// TIA Portal project "thuc_hanh_2" (V14)

(* hardware
DEVICE "S7-1200 station_1"  S7-1200 Station
   slot 0: "Rack_0"  S7-1200 Rack  Rack  V1.0
   slot 1: "PLC_1"  CPU 1214C DC/DC/DC  6ES7 214-1AG40-0XB0  V4.2
*)

// ===== PLC "PLC_1"  CPU 1214C DC/DC/DC =====

VAR_GLOBAL   // PLC tag table "Default tag table"
   "Tag_1" AT %M0.0 : Bool;
   "Tag_2" AT %Q0.0 : Bool;
   "enable" AT %M0.1 : Bool;
   "count_" AT %M0.2 : Bool;
   "reset_count" AT %M0.3 : Bool;
   "done_count" AT %M0.4 : Bool;
   "stop" AT %M0.5 : Bool;
   "Tag_3" AT %Q0.1 : Bool;
   "reset" AT %I0.0 : Bool;
   "start" AT %I0.1 : Bool;
   "Tag_4" AT %I0.3 : Bool;
END_VAR

// folder: System blocks/Program resources

DATA_BLOCK "IEC_Timer_0_DB"   // DB1
{ S7_Optimized_Access := 'TRUE' }
AUTHOR : Simatic
FAMILY : IEC
NAME : IEC_TMR
VERSION : 1.0
// stored: InstanceOfName IEC_TIMER
"IEC_TIMER"
BEGIN
END_DATA_BLOCK

DATA_BLOCK "IEC_Timer_0_DB_1"   // DB2
{ S7_Optimized_Access := 'TRUE' }
AUTHOR : Simatic
FAMILY : IEC
NAME : IEC_TMR
VERSION : 1.0
// stored: InstanceOfName IEC_TIMER
"IEC_TIMER"
BEGIN
END_DATA_BLOCK

DATA_BLOCK "IEC_Counter_0_DB"   // DB3
{ S7_Optimized_Access := 'TRUE' }
AUTHOR : Simatic
FAMILY : IEC
NAME : CNTR
VERSION : 1.0
// stored: InstanceOfName IEC_COUNTER
"IEC_COUNTER"
BEGIN
END_DATA_BLOCK

// folder: (top level)

ORGANIZATION_BLOCK "Main"   // OB1, LAD, ProgramCycle
TITLE = "Main Program Sweep (Cycle)"
{ S7_Optimized_Access := 'TRUE' }
VERSION : 0.1
   VAR_INPUT
      Initial_Call : Bool;   // Initial call of this OB
      Remanence : Bool;   // =True, if remanent data are available
   END_VAR
   VAR_TEMP
      count : Bool;
   END_VAR
BEGIN

REGION Network 1
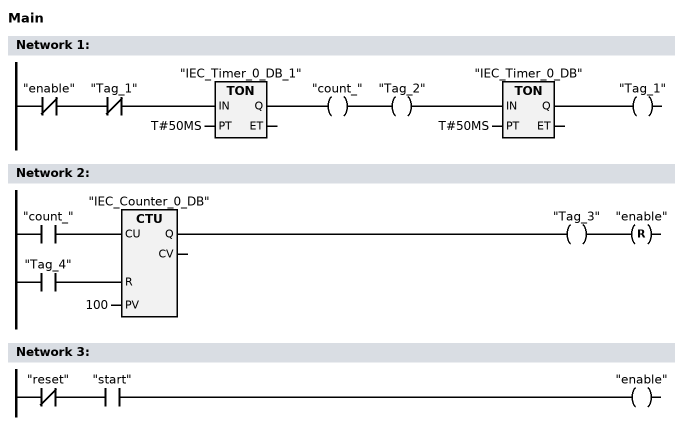
   "IEC_Timer_0_DB_1".TON(IN := NOT "enable" AND NOT "Tag_1", PT := T#50MS);
   "count_" := "IEC_Timer_0_DB_1".Q;
   "Tag_2" := "IEC_Timer_0_DB_1".Q;
   "IEC_Timer_0_DB".TON(IN := "IEC_Timer_0_DB_1".Q, PT := T#50MS);
   "Tag_1" := "IEC_Timer_0_DB".Q;
END_REGION

REGION Network 2
   "IEC_Counter_0_DB".CTU(CU := "count_", R := "Tag_4", PV := 100);
   "Tag_3" := "IEC_Counter_0_DB".Q;
   IF "IEC_Counter_0_DB".Q THEN "enable" := FALSE; END_IF;
END_REGION

REGION Network 3
   RUNG wire#powerrail
      I_Contact( "reset" )
      Contact( "start" )
      Coil( "enable" )
   END_RUNG
   // the same network as SCL:
   "enable" := NOT "reset" AND "start";
END_REGION
END_ORGANIZATION_BLOCK